// TIA Portal project "Week2_Ex1" (V14)

(* hardware
DEVICE "S7-1200 station_1"  S7-1200 Station
   slot 0: "Rack_0"  S7-1200 Rack  Rack  V1.0
   slot 1: "PLC_1"  CPU 1214C DC/DC/DC  6ES7 214-1AG40-0XB0  V4.2
*)

// ===== PLC "PLC_1"  CPU 1214C DC/DC/DC =====

VAR_GLOBAL   // PLC tag table "Default tag table"
   "Tag_1" AT %I0.7 : Bool;
   "Tag_2" AT %Q0.7 : Bool;
   "Tag_3" AT %Q1.0 : Bool;
   "Tag_4" AT %Q1.1 : Bool;
   "Tag_5" AT %I0.4 : Bool;
   "Tag_6" AT %I0.6 : Bool;
   "Tag_7" AT %I0.5 : Bool;
   "Tag_8" AT %I0.2 : Bool;
   "Tag_9" AT %I0.3 : Bool;
   "Tag_10" AT %I0.1 : Bool;
   "Tag_11" AT %M0.1 : Bool;
   "Tag_12" AT %M0.2 : Bool;
   "Tag_13" AT %M0.3 : Bool;
   "Tag_14" AT %M0.4 : Bool;
   "Tag_15" AT %M0.5 : Bool;
   "Tag_16" AT %M0.6 : Bool;
   "Tag_17" AT %M0.7 : Bool;
   "Tag_18" AT %MW10 : Int;
   "Tag_19" AT %MW11 : Int;
   "Tag_20" AT %MW12 : Int;
   "Tag_21" AT %MW13 : Int;
   "Tag_22" AT %MW14 : Word;
   "Tag_23" AT %MW15 : Int;
   "Tag_24" AT %MW16 : Word;
   "Tag_25" AT %MW17 : Int;
END_VAR

// folder: System blocks/Program resources

DATA_BLOCK "IEC_Timer_0_DB"   // DB1
{ S7_Optimized_Access := 'TRUE' }
AUTHOR : Simatic
FAMILY : IEC
NAME : IEC_TMR
VERSION : 1.0
// stored: InstanceOfName IEC_TIMER
"IEC_TIMER"
BEGIN
END_DATA_BLOCK

DATA_BLOCK "IEC_Timer_0_DB_1"   // DB2
{ S7_Optimized_Access := 'TRUE' }
AUTHOR : Simatic
FAMILY : IEC
NAME : IEC_TMR
VERSION : 1.0
// stored: InstanceOfName IEC_TIMER
"IEC_TIMER"
BEGIN
END_DATA_BLOCK

// folder: (top level)

ORGANIZATION_BLOCK "Main"   // OB1, LAD, ProgramCycle
TITLE = "Main Program Sweep (Cycle)"
{ S7_Optimized_Access := 'TRUE' }
VERSION : 0.1
   VAR_INPUT
      Initial_Call : Bool;   // Initial call of this OB
      Remanence : Bool;   // =True, if remanent data are available
   END_VAR
BEGIN

REGION Network 1
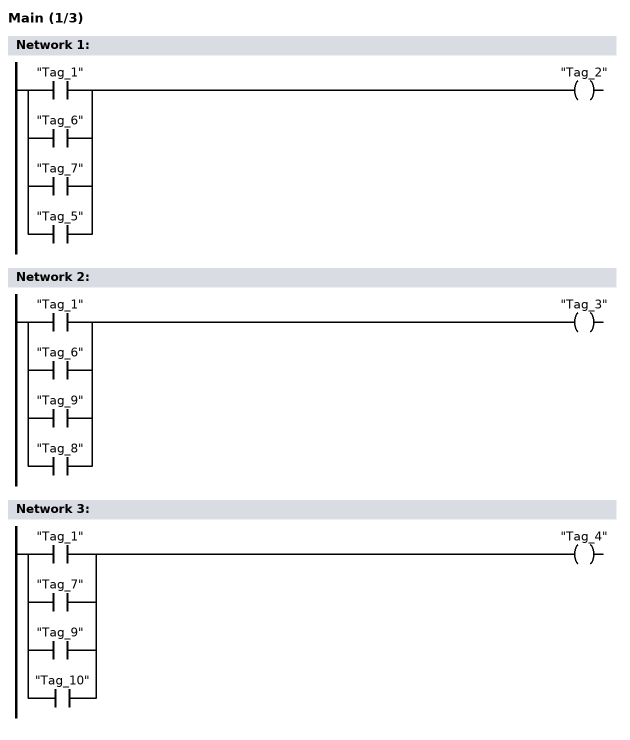
   RUNG wire#powerrail
      Contact( "Tag_1" )
      wire#w1
      Coil( "Tag_2" )
   END_RUNG
   RUNG wire#powerrail
      Contact( "Tag_6" )
   END_RUNG wire#w1
   RUNG wire#powerrail
      Contact( "Tag_7" )
   END_RUNG wire#w1
   RUNG wire#powerrail
      Contact( "Tag_5" )
   END_RUNG wire#w1
   // the same network as SCL:
   "Tag_2" := "Tag_1" OR "Tag_6" OR "Tag_7" OR "Tag_5";
END_REGION

REGION Network 2
   RUNG wire#powerrail
      Contact( "Tag_1" )
      wire#w1
      Coil( "Tag_3" )
   END_RUNG
   RUNG wire#powerrail
      Contact( "Tag_6" )
   END_RUNG wire#w1
   RUNG wire#powerrail
      Contact( "Tag_9" )
   END_RUNG wire#w1
   RUNG wire#powerrail
      Contact( "Tag_8" )
   END_RUNG wire#w1
   // the same network as SCL:
   "Tag_3" := "Tag_1" OR "Tag_6" OR "Tag_9" OR "Tag_8";
END_REGION

REGION Network 3
   RUNG wire#powerrail
      Contact( "Tag_1" )
      wire#w1
      Coil( "Tag_4" )
   END_RUNG
   RUNG wire#powerrail
      Contact( "Tag_7" )
   END_RUNG wire#w1
   RUNG wire#powerrail
      Contact( "Tag_9" )
   END_RUNG wire#w1
   RUNG wire#powerrail
      Contact( "Tag_10" )
   END_RUNG wire#w1
   // the same network as SCL:
   "Tag_4" := "Tag_1" OR "Tag_7" OR "Tag_9" OR "Tag_10";
END_REGION

REGION Network 4
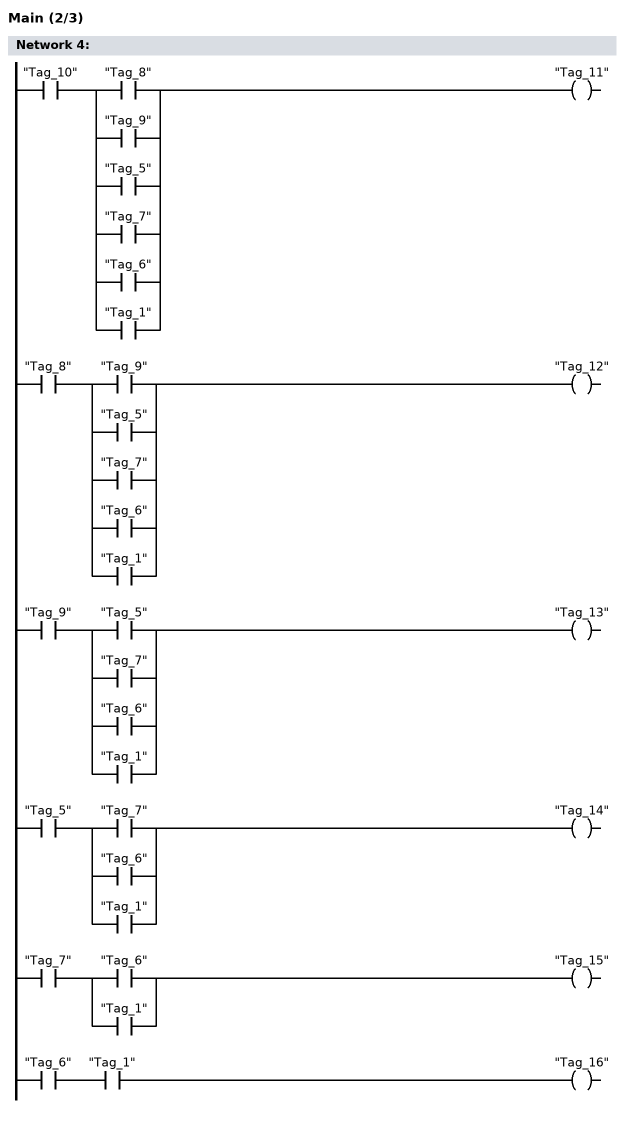
   RUNG wire#powerrail
      Contact( "Tag_10" )
      wire#w1
      Contact( "Tag_8" )
      wire#w2
      Coil( "Tag_11" )
   END_RUNG
   RUNG wire#w1
      Contact( "Tag_9" )
   END_RUNG wire#w2
   RUNG wire#w1
      Contact( "Tag_5" )
   END_RUNG wire#w2
   RUNG wire#w1
      Contact( "Tag_7" )
   END_RUNG wire#w2
   RUNG wire#w1
      Contact( "Tag_6" )
   END_RUNG wire#w2
   RUNG wire#w1
      Contact( "Tag_1" )
   END_RUNG wire#w2
   RUNG wire#powerrail
      Contact( "Tag_8" )
      wire#w3
      Contact( "Tag_9" )
      wire#w4
      Coil( "Tag_12" )
   END_RUNG
   RUNG wire#w3
      Contact( "Tag_5" )
   END_RUNG wire#w4
   RUNG wire#w3
      Contact( "Tag_7" )
   END_RUNG wire#w4
   RUNG wire#w3
      Contact( "Tag_6" )
   END_RUNG wire#w4
   RUNG wire#w3
      Contact( "Tag_1" )
   END_RUNG wire#w4
   RUNG wire#powerrail
      Contact( "Tag_9" )
      wire#w5
      Contact( "Tag_5" )
      wire#w6
      Coil( "Tag_13" )
   END_RUNG
   RUNG wire#w5
      Contact( "Tag_7" )
   END_RUNG wire#w6
   RUNG wire#w5
      Contact( "Tag_6" )
   END_RUNG wire#w6
   RUNG wire#w5
      Contact( "Tag_1" )
   END_RUNG wire#w6
   RUNG wire#powerrail
      Contact( "Tag_5" )
      wire#w7
      Contact( "Tag_7" )
      wire#w8
      Coil( "Tag_14" )
   END_RUNG
   RUNG wire#w7
      Contact( "Tag_6" )
   END_RUNG wire#w8
   RUNG wire#w7
      Contact( "Tag_1" )
   END_RUNG wire#w8
   RUNG wire#powerrail
      Contact( "Tag_7" )
      wire#w9
      Contact( "Tag_6" )
      wire#w10
      Coil( "Tag_15" )
   END_RUNG
   RUNG wire#w9
      Contact( "Tag_1" )
   END_RUNG wire#w10
   RUNG wire#powerrail
      Contact( "Tag_6" )
      Contact( "Tag_1" )
      Coil( "Tag_16" )
   END_RUNG
   // the same network as SCL:
   "Tag_11" := "Tag_10" AND ("Tag_8" OR "Tag_9" OR "Tag_5" OR "Tag_7" OR "Tag_6" OR "Tag_1");
   "Tag_12" := "Tag_8" AND ("Tag_9" OR "Tag_5" OR "Tag_7" OR "Tag_6" OR "Tag_1");
   "Tag_13" := "Tag_9" AND ("Tag_5" OR "Tag_7" OR "Tag_6" OR "Tag_1");
   "Tag_14" := "Tag_5" AND ("Tag_7" OR "Tag_6" OR "Tag_1");
   "Tag_15" := "Tag_7" AND ("Tag_6" OR "Tag_1");
   "Tag_16" := "Tag_6" AND "Tag_1";
END_REGION

REGION Network 5
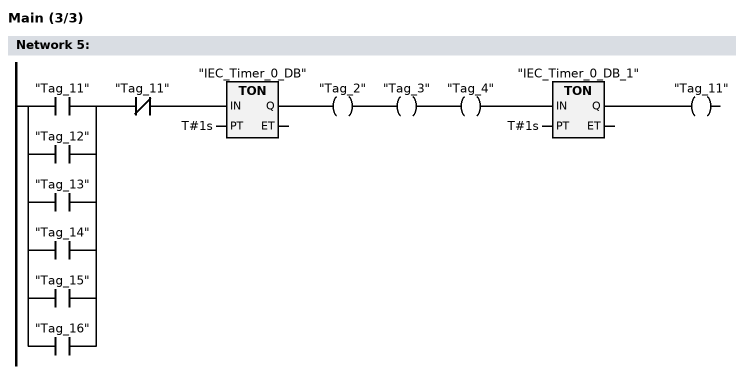
   "IEC_Timer_0_DB".TON(IN := ("Tag_11" OR "Tag_12" OR "Tag_13" OR "Tag_14" OR "Tag_15" OR "Tag_16") AND NOT "Tag_11",
                        PT := T#1s);
   "Tag_2" := "IEC_Timer_0_DB".Q;
   "Tag_3" := "IEC_Timer_0_DB".Q;
   "Tag_4" := "IEC_Timer_0_DB".Q;
   "IEC_Timer_0_DB_1".TON(IN := "IEC_Timer_0_DB".Q, PT := T#1s);
   "Tag_11" := "IEC_Timer_0_DB_1".Q;
END_REGION
END_ORGANIZATION_BLOCK